FUNCTION_BLOCK MovementBlockType1 (* Protection layer *)
  (* Standard: 61499-2 *)
  (* Version 1.0, 2008-11-09, Cheng Pang, The University of Auckland, Stable build. *)
  (* Compiler header: package fb.rt.pnp; *)
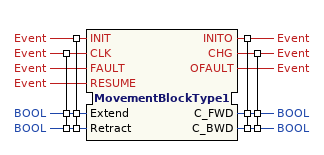
  EVENT_INPUT
    INIT WITH Extend, Retract; (* Initialization Request *)
    CLK WITH Extend, Retract; (* Clock signal *)
    FAULT;
    RESUME;
  END_EVENT
  EVENT_OUTPUT
    INITO WITH C_FWD, C_BWD; (* Initialization Confirm *)
    CHG WITH C_FWD, C_BWD; (* Data outputs changed *)
    OFAULT;
  END_EVENT
  VAR_INPUT
    Extend : BOOL; (* Move forwards *)
    Retract : BOOL; (* Move backwards *)
  END_VAR
  VAR_OUTPUT
    C_FWD : BOOL; (* Confirmed move forwards *)
    C_BWD : BOOL; (* Confirmed move backwards *)
  END_VAR
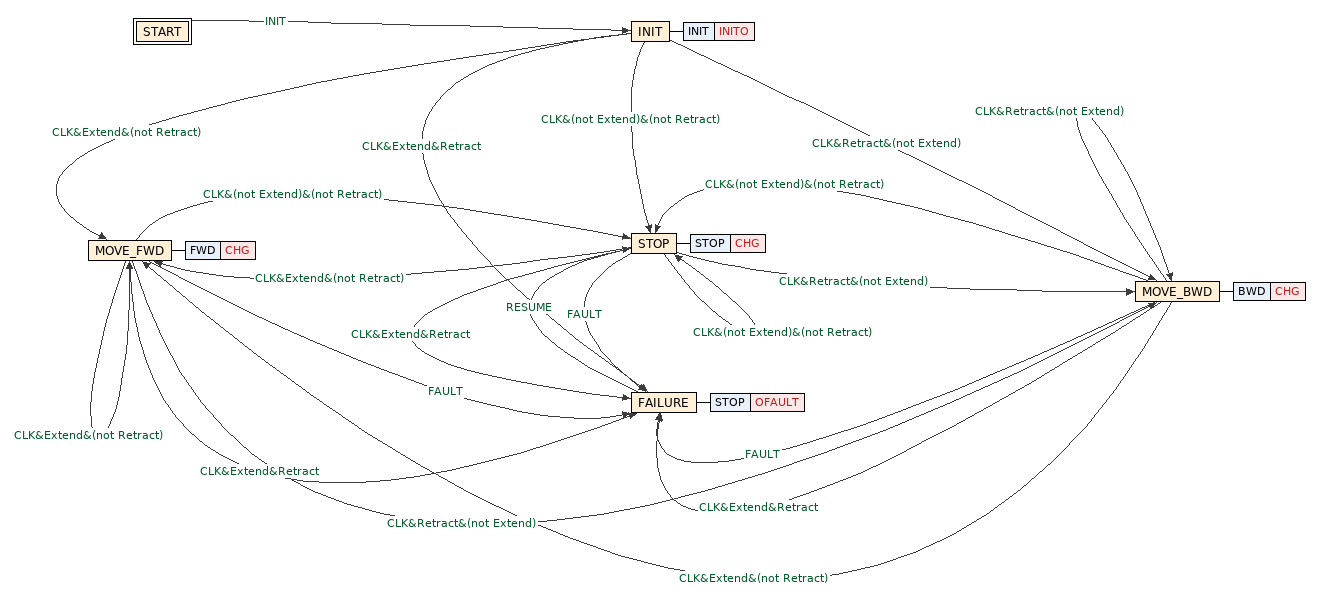
  EC_STATES
    START; (* Initial State *)
    INIT : INIT -> INITO; (* Initialization *)
    MOVE_FWD : FWD -> CHG;
    MOVE_BWD : BWD -> CHG;
    STOP : STOP -> CHG;
    FAILURE : STOP -> OFAULT;
  END_STATES
  EC_TRANSITIONS
    START TO INIT := INIT;
    INIT TO MOVE_FWD := CLK&Extend&(not Retract);
    INIT TO STOP := CLK&(not Extend)&(not Retract);
    INIT TO MOVE_BWD := CLK&Retract&(not Extend);
    MOVE_FWD TO FAILURE := FAULT;
    STOP TO FAILURE := FAULT;
    MOVE_BWD TO FAILURE := FAULT;
    MOVE_FWD TO STOP := CLK&(not Extend)&(not Retract);
    MOVE_BWD TO STOP := CLK&(not Extend)&(not Retract);
    STOP TO MOVE_FWD := CLK&Extend&(not Retract);
    STOP TO MOVE_BWD := CLK&Retract&(not Extend);
    FAILURE TO STOP := RESUME;
    MOVE_FWD TO MOVE_BWD := CLK&Retract&(not Extend);
    MOVE_BWD TO MOVE_FWD := CLK&Extend&(not Retract);
    STOP TO FAILURE := CLK&Extend&Retract;
    INIT TO FAILURE := CLK&Extend&Retract;
    MOVE_FWD TO FAILURE := CLK&Extend&Retract;
    MOVE_BWD TO FAILURE := CLK&Extend&Retract;
    MOVE_FWD TO MOVE_FWD := CLK&Extend&(not Retract);
    MOVE_BWD TO MOVE_BWD := CLK&Retract&(not Extend);
    STOP TO STOP := CLK&(not Extend)&(not Retract);
  END_TRANSITIONS
  ALGORITHM INIT IN Java: (* Initialization algorithm *)
C_FWD.value = false;
C_BWD.value = false;
  END_ALGORITHM
  ALGORITHM FWD IN Java: (* Normally executed algorithm *)
C_FWD.value = true;
C_BWD.value = false;
//System.out.println("\n  MotionLogic.FWD:");
//System.out.println("  Moving forwards");
  END_ALGORITHM
  ALGORITHM BWD IN Java:
C_FWD.value = false;
C_BWD.value = true;

//System.out.println("Moving Backwards");
  END_ALGORITHM
  ALGORITHM STOP IN Java:
C_FWD.value = false;
C_BWD.value = false;

//System.out.println("Stopped");
  END_ALGORITHM
END_FUNCTION_BLOCK
